Fanuc KAREL source: kf00079.KL

-- PROVISIONAL review KL for V770-1; original PC SHA256 49419a5a232205485fa8769843a75aab20b6520bf12b1b39ed760fc161f1f2a6
-- Incomplete behavior may be omitted. Consult companion uncertainty JSON. Do not deploy.
PROGRAM KF00079
%NOLOCKGROUP
BEGIN
  -- UNRESOLVED_PC offsets 5-15; opcodes 3F,75
  -- UNRESOLVED_PC offsets 20-29; opcodes 3F,75
  -- UNRESOLVED_PC offsets 34-45; opcodes 2E,23
  -- UNRESOLVED_PC offsets 50-61; opcodes 2E,23
  -- UNRESOLVED_PC offsets 66-84; opcodes 27,22,2A,22,31
  -- UNRESOLVED_PC offsets 89-93; opcodes 7F
END KF00079
